FUNCTION_BLOCK FB_TcUnitExample EXTENDS FB_TestSuite
VAR
	hr				: HRESULT;		
	fbTcUnitAdapter : FB_TcUnitAdapter;
	
	stActual		: ST_DemoDataType;
	{attribute 'analysis' := '-33'}
	stResult		: ST_VerificationResult;
END_VAR

TEST('Test some stuff with TcHaxx.Snappy');

// ARRANGE

// ACT
stActual := F_CreateDemoData();

// ASSERT
hr := fbTcUnitAdapter.Verify(anyArg:= stActual);

IF NOT PENDING(hr) THEN
	TEST_FINISHED_NAMED('Test some stuff with TcHaxx.Snappy');
END_IF

END_FUNCTION_BLOCK

(* stored: Version 1.1.0.1, ProductVersion 3.1.4026.18
   POU FB_TcUnitExample: Id {2328aed7-3c8d-44a5-a37e-d87d39d21ab0}, SpecialFunc None *)
